FUNCTION_BLOCK FB_Tracking
VAR_IN_OUT
	stAxis  : ARRAY [GVL.cXP .. GVL.cXM] OF ST_AxisGroup;	
END_VAR
VAR_INPUT
	eCommand 			: E_Commands;
	bMotionDone			: BOOL;
	inReset				: ST_Reset;
	inMoveAxisAbsolute	: ST_MoveAxisAbsolute;
	inMoveAxisRelative	: ST_MoveAxisRelative;
END_VAR
VAR_OUTPUT
	stOutMotionDone : ST_MotionDone;
END_VAR
VAR
	//used in tracking Action
	stTrack			: ARRAY [0 .. 4] OF ST_TRACK;
	stTrackTemp		: ST_TRACK;  // Used for the sorting of stTrack.
	keepSorting		: BOOL;      // Used for the sorting.
	bGoNextSeq		: BOOL;
	nAxisID			: INT;
	nMask			: ULINT := 16#FFFF_FFFF_0000_0000;
	
	//used in determining target duration
	fSpeed			: LREAL;
	tTargetDur		: LTIME;
	fDistance		: LREAL;
	
	fbMoving_Rtrig : ARRAY[0 .. 1] OF R_TRIG;
	fbRtrig		: ARRAY[GVL.cHallLower..GVL.cHallUpper] OF R_Trig;
	bInMotion	: BOOL;
	stMotionDone : ARRAY [0..1] OF ST_MotionDone;	
	nSequence	: DINT;
	nLastMoved	: INT;
	
	//counter
	i, j, k, m		: INT := 0;
	nTPC	: INT; //Trip Per Cycle

	// Save task-start and MIO SysTime values in a ring buffer x of depth N. The newest
	// entry is x[i], the oldest is x[(i + 1) mod N], assuming that the buffer is full.
	iTimeBuffer: INT := GVL.cTimeBufferDepth - 1;
	taskStartExtTime: T_TaskStartTimes;
	mioSysTime: T_MioSysTimes;

END_VAR

//////////////////////////////////////////////////////////////
// Call this function block once per cycle to process any updated information about blade set motion and send updates to CCS if required.
//////////////////////////////////////////////////////////////

// Update some times for the previous and current cycles.
iTimeBuffer := (iTimeBuffer + 1) MOD GVL.cTimeBufferDepth;
taskStartExtTime[iTimeBuffer] := F_GetCurExtTime64(GVL.DcToExtTimeOffset, GVL.DcToTcTimeOffset);
mioSysTime[iTimeBuffer] := GVL.mioSysTime;

stAxis[GVL.cXP].bTrackedFlag:=FALSE;
stAxis[GVL.cXM].bTrackedFlag:=FALSE;
nTPC:=0;

// Detect start of motion for the +X blade set, rising edge of its Moving flag from the motor controller.
// Reset motion profile parameters in a local motion-done message not monitored by CCS.
fbMoving_Rtrig[GVL.cXP](CLK:=stAxis[GVL.cXP].axisRef.Status.Moving);
IF fbMoving_Rtrig[GVL.cXP].Q THEN
	// Prepare to record motion profile information.
	bInMotion:=TRUE;  // We're moving!
	stMotionDone[GVL.cXP].axisNum := GVL.cXP; // Axis is +X.
	stMotionDone[GVL.cXP].nsamples := 0;      // No encoder samples yet.
	stMotionDone[GVL.cXP].ntrans := 0;        // No Hall transitions yet.
	stMotionDone[gvl.cXP].startPos := stAxis[GVL.cXP].axisRef.NcToPlc.ActPos;   // Where are we now?
	stMotionDone[GVL.cXP].startTime := taskStartExtTime[iTimeBuffer];
	stMotionDone[GVL.cXP].targetDur := LTIME#0D0H0M0S0MS0US0NS;  // Don't know yet how long this motion will take.
END_IF

// The same, but for the -X blade set.
fbMoving_Rtrig[GVL.cXM](CLK:=stAxis[GVL.cXM].axisRef.Status.Moving);
IF fbMoving_Rtrig[GVL.cXM].Q THEN
	// Prepare to record motion profile information.
	bInMotion:=TRUE;
	stMotionDone[gvl.cXM].axisNum := GVL.cXM;
	stMotionDone[gvl.cXM].nsamples := 0;
	stMotionDone[gvl.cXM].ntrans := 0;
	stMotionDone[gvl.cXM].startPos := stAxis[GVL.cXM].axisRef.NcToPlc.ActPos;
	stMotionDone[gvl.cXM].startTime := taskStartExtTime[iTimeBuffer];
	stMotionDone[gvl.cXM].targetDur := LTIME#0D0H0M0S0MS0US0NS;
END_IF

// Assuming that a motion command was issued by CCS, calculate how long the motion is supposed to last.
// Output is tTargetDur.
IF eCommand = E_Commands.takeExposure THEN
	fSpeed	:= inReset.speed;   // Speed from reset command (actually now set elsewhere in this PLC code).
	IF (fSpeed>0) THEN
		IF (fSpeed>1668.355556) THEN
			fSpeed:=1668.355556;
		END_IF
		tTargetDur 	:= LREAL_TO_LTIME((2*GVL.cPosEnd)/(fSpeed)*EXPT(10,9));
	END_IF
ELSIF eCommand = E_Commands.moveAxisAbsolute THEN
	// MoveAxisAbsolute message contains target position and speed of motion.
	fDistance := ABS(stAxis[inMoveAxisAbsolute.axisIndex].axisRef.NcToPlc.ActPos - inMoveAxisAbsolute.position);
	fSpeed	:= inMoveAxisAbsolute.speed;
	IF (fSpeed>0) THEN
		IF (fSpeed>1668.355556) THEN
			fSpeed:=1668.355556;
		END_IF
		tTargetDur 	:= LREAL_TO_LTIME(((2*fDistance)/(fSpeed))*EXPT(10,9));
	END_IF
ELSIF eCommand = E_Commands.moveAxisRelative THEN
	// MoveAxisRelative message contains position change and how long to take to do it.
	tTargetDur	:= TIME_TO_LTIME(inMoveAxisRelative.moveTime);
END_IF

//Checks to see which blade set last started moving.
IF (stAxis[GVL.cXM].axisRef.Status.Moving AND stAxis[GVL.cXP].axisRef.Status.InTargetPosition) THEN
	nLastMoved:=GVL.cXM;
ELSIF (stAxis[GVL.cXP].axisRef.Status.Moving AND stAxis[GVL.cXM].axisRef.Status.InTargetPosition) THEN
	nLastMoved:=GVL.cXP;
END_IF

////////// Handle the completion of a blade set motion. //////////
IF bMotionDone THEN
	//use for determining which blade set has finished during a travelling slit motion
	IF (stAxis[GVL.cXM].axisRef.Status.Moving AND stAxis[GVL.cXP].axisRef.Status.InTargetPosition) THEN
		nAxisID:=GVL.cXP;
	ELSIF (stAxis[GVL.cXP].axisRef.Status.Moving AND stAxis[GVL.cXM].axisRef.Status.InTargetPosition) THEN
		nAxisID:=GVL.cXM;
	ELSE 
		nAxisID:=nLastMoved;
	END_IF
	//bInMotion flag remains true if either of the blade sets is still in motion
	IF ((NOT stAxis[GVL.cXP].axisRef.Status.Moving) AND (NOT stAxis[GVL.cXM].axisRef.Status.Moving)) THEN
		bInMotion := FALSE;
	END_IF
	// Complete our local motion-done message.
	nSequence := nSequence+1;
	// The motor controller doesn't report exactly when motion was completed, so we assume that it was when the process data
	// from the controller reached us, i.e., at the start of the current cycle.
	stMotionDone[nAxisID].actualDur := ULINT_TO_LTIME(taskStartExtTime[iTimeBuffer] - stMotionDone[nAxisID].startTime);
	stMotionDone[nAxisID].targetDur := tTargetDur;
	stMotionDone[nAxisID].targetPos := stAxis[nAxisID].axisRef.NcToPlc.TargetPos;
	stMotionDone[nAxisID].endPos := stAxis[nAxisID].axisRef.NcToPlc.ActPos;
	stMotionDone[nAxisId].ptpState := MAIN.ptpDiagInfo.PTPState;
	stMotionDone[nAxisId].leapSeconds := MAIN.ptpDiagInfo.CurrentUtcOffset;
	stMotionDone[nAxisId].leapIsValid := TO_BOOL(MAIN.ptpDiagInfo.CurrentUtcOffsetIsValid);
	// Copy our local motion-done message to the location that's monitored by CCS.
	stOutMotionDone:=stMotionDone[nAxisID];
	stOutMotionDone.sequence:=nSequence;  // Ensure message gets sent to CCS by making sure that at least one field has a changed value.
END_IF


////////// Collect information on any Hall switch transitions from the MIOs. //////////
// nNumOfINputs[i] is linked to the event count for the MIO channel assigned to Hall sensor i.
// bInputEventState[i] is linked to the current MIO channel state for Hall sensor i.
// nInputEventTime[i] is linked to the first transition timestamp for Hall sensor i. We assume there is at most one per cycle per channel, though
// more than one channel may have a timestamp available in the same cycle.
// New timestamps are added to the end of the stTrack array.

FOR i:=GVL.cHallLower TO GVL.cHallUpper BY 1 DO
	fbRtrig[i](CLK:=GVL.nNumOfInputs[i].0);  // Look for a rising edge in channel status, which means we have a transition timestamp.
	IF fbRtrig[i].Q THEN
		stTrack[nTPC].nSeqToCompare := INT_TO_WORD((i*10)+5);
		stTrack[nTPC].bEdgeToCompare := GVL.bInputEventState[i];
		stTrack[nTPC].nHallID := i;
		stTrack[nTPC].tScanTime := 
			F_MioExtTime(i, GVL.nInputEventTime[i], iTimeBuffer, taskStartExtTime, mioSysTime);  // ADC timestamp -> ext time.
 		// Count the number of entries stored in stTrack.
		nTPC:=nTPC+1;
	END_IF
END_FOR
	
// Calibration stores events in time order, and later code that assigns locations to Hall events requires
// exactly the same ordering for a given blade set and direction of motion. If during this cycle we picked up
// events from more than one channel we'll have to sort them by time. At most a handful of events
// may occur in a cycle so an exchange sort will do.
IF nTPC > 1 THEN
	keepSorting := TRUE;  // Do we need to keep sorting?
	WHILE keepSorting DO
		keepSorting := FALSE;
		FOR j:= nTPC - 1 TO 1 BY -1 DO
			IF (stTrack[j].tScanTime < stTrack[j-1].tScanTime) THEN  // Use <, not <=, to make it a stable sort.
				stTrackTemp := stTrack[j];
				stTrack[j] := stTrack[j-1];
				stTrack[j-1] := stTrackTemp;
				keepSorting := TRUE;  // Need to keep sorting if an exchange was made.
			END_IF
		END_FOR
	END_WHILE
END_IF


// If we picked up some Hall transitions this cycle, then we need to take position samples (encoder readout).
// We want to check if the position of a blade set at the time of a Hall transition agrees with the
// Hall switch position taken from the last calibration.
IF nTPC>0 THEN
	FOR k:=0 TO nTPC-1 BY 1 DO
		IF (stAxis[GVL.cXP].axisRef.Status.Moving AND stAxis[GVL.cXM].axisRef.Status.Moving) AND
			(stAxis[GVL.cXP].axisRef.Status.PositiveDirection AND stAxis[GVL.cXM].axisRef.Status.PositiveDirection) THEN
			ACT_TrackingDoublePositive();
		ELSIF (stAxis[GVL.cXP].axisRef.Status.Moving AND stAxis[GVL.cXM].axisRef.Status.Moving) AND
			(stAxis[GVL.cXP].axisRef.Status.NegativeDirection AND stAxis[GVL.cXM].axisRef.Status.NegativeDirection) THEN
			ACT_TrackingDoubleNegative();
		ELSE
			ACT_TrackingSingle();
		END_IF
		bGoNextSeq:=FALSE;
	END_FOR
END_IF

ACTION ACT_TrackingDoubleNegative:
// Take encoder samples and compare against Hall transitions when both blade sets are moving toward decreasing camera X coordinate.
// Remember, this code is being called from inside a loop over the contents of stTrack[] with k being the loop variable.
// We have to first assign a Hall event to a blade set before we can find out the motion start times and
// calculate elapsed times from that. 

// +X blade set
IF stAxis[GVL.cXP].axisRef.Status.Moving THEN
	//Compare current sequence with recorded sequence. Update position if match. Negative direction.
	IF stAxis[GVL.cXP].axisRef.status.NegativeDirection AND stAxis[GVL.cXP].stHall[GVL.cDirNeg, stAxis[GVL.cXP].nTripCount].nSeq = stTrack[k].nSeqToCompare AND
			stAxis[GVL.cXP].stHall[GVL.cDirNeg, stAxis[GVL.cXP].nTripCount].bEdge = stTrack[k].bEdgeToCompare AND (NOT bGoNextSeq) THEN
		stAxis[GVL.cXP].fHallPosAct := stAxis[GVL.cXP].fHallPosCal[GVL.cDirNeg, stAxis[GVL.cXP].nTripCount];
		stAxis[GVL.cXP].nTripCount := stAxis[GVL.cXP].nTripCount - 1;		
		//track difference between hall sensor and encoder data at trip point
		stAxis[GVL.cXP].fPosDiffAtTrip := stAxis[GVL.cXP].axisRef.NcToPlc.ActPos - stAxis[GVL.cXP].fHallPosAct;
		stAxis[GVL.cXP].bTrackedFlag:=TRUE;
		bGoNextSeq:=TRUE;
		
		IF bInMotion AND MAIN.outShutterStatus.smState<>E_StatesMaint.Calibrating THEN
			nAxisID := GVL.cXP;
			// The Hall event belongs to the +X blade set.
			stMotionDone[GVL.cXP].trans[stMotionDone[GVL.cXP].ntrans].extTime := stTrack[k].tScanTime;
			stMotionDone[GVL.cXP].trans[stMotionDone[GVL.cXP].ntrans].id := stTrack[k].nHallID;
			stMotionDone[GVL.cXP].trans[stMotionDone[GVL.cXP].ntrans].on := stTrack[k].bEdgeToCompare;
			stMotionDone[GVL.cXP].trans[stMotionDone[GVL.cXP].ntrans].pos := stAxis[GVL.cXP].fHallPosAct;
			stMotionDone[GVL.cXP].ntrans := stMotionDone[GVL.cXP].ntrans +1;
			// We're taking the encoder value from process data for this cycle, so the closest
			// approximation we have to the actual sample time is the time at the start of the cycle.
			stMotionDone[GVL.cXP].samples[stMotionDone[GVL.cXP].nsamples].extTime := taskStartExtTime[iTimeBuffer];
			stMotionDone[GVL.cXP].samples[stMotionDone[GVL.cXP].nsamples].pos := stAxis[GVL.cXP].axisRef.NcToPlc.ActPos;
			stMotionDone[GVL.cXP].nsamples := stMotionDone[GVL.cXP].nsamples + 1;
		END_IF
		
	END_IF
END_IF

// -X blade set
IF stAxis[GVL.cXM].axisRef.Status.Moving THEN
	//Compare current sequence with recorded sequence. Update position if match. Negative direction.
	IF stAxis[GVL.cXM].axisRef.status.NegativeDirection AND stAxis[GVL.cXM].stHall[GVL.cDirNeg, stAxis[GVL.cXM].nTripCount].nSeq = stTrack[k].nSeqToCompare AND
			stAxis[GVL.cXM].stHall[GVL.cDirNeg, stAxis[GVL.cXM].nTripCount].bEdge = stTrack[k].bEdgeToCompare AND (NOT bGoNextSeq) THEN
		stAxis[GVL.cXM].fHallPosAct := stAxis[GVL.cXM].fHallPosCal[GVL.cDirNeg, stAxis[GVL.cXM].nTripCount];
		stAxis[GVL.cXM].nTripCount := stAxis[GVL.cXM].nTripCount + 1;	
		//track difference between hall sensor and encoder data at trip point
		stAxis[GVL.cXM].fPosDiffAtTrip := stAxis[GVL.cXM].axisRef.NcToPlc.ActPos - stAxis[GVL.cXM].fHallPosAct;
		stAxis[GVL.cXM].bTrackedFlag:=TRUE;
		bGoNextSeq:=TRUE;
		
		IF bInMotion AND MAIN.outShutterStatus.smState<>E_StatesMaint.Calibrating THEN
			nAxisID:= GVL.cXM;
			// The Hall event belongs to the -X blade set.
			stMotionDone[GVL.cXM].trans[stMotionDone[GVL.cXM].ntrans].extTime := stTrack[k].tScanTime;
			stMotionDone[GVL.cXM].trans[stMotionDone[GVL.cXM].ntrans].id := stTrack[k].nHallID;
			stMotionDone[GVL.cXM].trans[stMotionDone[GVL.cXM].ntrans].on := stTrack[k].bEdgeToCompare;
			stMotionDone[GVL.cXM].trans[stMotionDone[GVL.cXM].ntrans].pos := stAxis[GVL.cXM].fHallPosAct;
			stMotionDone[GVL.cXM].ntrans := stMotionDone[GVL.cXM].ntrans +1;

			stMotionDone[GVL.cXM].samples[stMotionDone[GVL.cXM].nsamples].extTime := taskStartExtTime[iTimeBuffer];
			stMotionDone[GVL.cXM].samples[stMotionDone[GVL.cXM].nsamples].pos := stAxis[GVL.cXM].axisRef.NcToPlc.ActPos;
			stMotionDone[GVL.cXM].nsamples := stMotionDone[GVL.cXM].nsamples + 1;
		END_IF
		
	END_IF
END_IF
END_ACTION

ACTION ACT_TrackingDoublePositive:
// Take encoder samples and compare against Hall transitions when both blade sets are moving toward increasing camera X coordinate.

// -X blade set
IF stAxis[GVL.cXM].axisRef.Status.Moving THEN
	//Compare current sequence with recorded sequence. Update position if match. Positive direction.
	IF stAxis[GVL.cXM].axisRef.status.PositiveDirection AND stAxis[GVL.cXM].stHall[GVL.cDirPos, stAxis[GVL.cXM].nTripCount].nSeq = stTrack[k].nSeqToCompare AND
			stAxis[GVL.cXM].stHall[GVL.cDirPos, stAxis[GVL.cXM].nTripCount].bEdge = stTrack[k].bEdgeToCompare AND (NOT bGoNextSeq) THEN
		stAxis[GVL.cXM].fHallPosAct := stAxis[GVL.cXM].fHallPosCal[GVL.cDirPos, stAxis[GVL.cXM].nTripCount];
		stAxis[GVL.cXM].nTripCount := stAxis[GVL.cXM].nTripCount - 1;	
		//track difference between hall sensor and encoder data at trip point
		stAxis[GVL.cXM].fPosDiffAtTrip := stAxis[GVL.cXM].axisRef.NcToPlc.ActPos - stAxis[GVL.cXM].fHallPosAct;
		stAxis[GVL.cXM].bTrackedFlag:=TRUE;
		bGoNextSeq:=TRUE;
		
		IF bInMotion AND MAIN.outShutterStatus.smState<>E_StatesMaint.Calibrating THEN
			nAxisID:= GVL.cXM;
			// The Hall event belongs to the -X blade set.
			stMotionDone[GVL.cXM].trans[stMotionDone[GVL.cXM].ntrans].extTime := stTrack[k].tScanTime;
			stMotionDone[GVL.cXM].trans[stMotionDone[GVL.cXM].ntrans].id := stTrack[k].nHallID;
			stMotionDone[GVL.cXM].trans[stMotionDone[GVL.cXM].ntrans].on := stTrack[k].bEdgeToCompare;
			stMotionDone[GVL.cXM].trans[stMotionDone[GVL.cXM].ntrans].pos := stAxis[GVL.cXM].fHallPosAct;
			stMotionDone[GVL.cXM].ntrans := stMotionDone[GVL.cXM].ntrans +1;
			
			stMotionDone[GVL.cXM].samples[stMotionDone[GVL.cXM].nsamples].extTime := taskStartExtTime[iTimeBuffer];
			stMotionDone[GVL.cXM].samples[stMotionDone[GVL.cXM].nsamples].pos := stAxis[GVL.cXM].axisRef.NcToPlc.ActPos;
			stMotionDone[GVL.cXM].nsamples := stMotionDone[GVL.cXM].nsamples + 1;
		END_IF
		
	END_IF
END_IF

// +X blade set
IF stAxis[GVL.cXP].axisRef.Status.Moving THEN
	//Compare current sequence with recorded sequence. Update position if match. Positive direction.
	IF stAxis[GVL.cXP].axisRef.status.PositiveDirection AND stAxis[GVL.cXP].stHall[GVL.cDirPos, stAxis[GVL.cXP].nTripCount].nSeq = stTrack[k].nSeqToCompare AND 
			stAxis[GVL.cXP].stHall[GVL.cDirPos, stAxis[GVL.cXP].nTripCount].bEdge = stTrack[k].bEdgeToCompare AND (NOT bGoNextSeq) THEN
		stAxis[GVL.cXP].fHallPosAct := stAxis[GVL.cXP].fHallPosCal[GVL.cDirPos, stAxis[GVL.cXP].nTripCount];
		stAxis[GVL.cXP].nTripCount := stAxis[GVL.cXP].nTripCount + 1;
		//track difference between hall sensor and encoder data at trip point
		stAxis[GVL.cXP].fPosDiffAtTrip := stAxis[GVL.cXP].axisRef.NcToPlc.ActPos - stAxis[GVL.cXP].fHallPosAct;
		stAxis[GVL.cXP].bTrackedFlag:=TRUE;
		bGoNextSeq:=TRUE;
		
		IF bInMotion AND MAIN.outShutterStatus.smState<>E_StatesMaint.Calibrating THEN
			nAxisID:= GVL.cXP;
			// The Hall event belongs to the +X blade set.
			stMotionDone[GVL.cXP].trans[stMotionDone[GVL.cXP].ntrans].extTime := stTrack[k].tScanTime;
			stMotionDone[GVL.cXP].trans[stMotionDone[GVL.cXP].ntrans].id := stTrack[k].nHallID;
			stMotionDone[GVL.cXP].trans[stMotionDone[GVL.cXP].ntrans].on := stTrack[k].bEdgeToCompare;
			stMotionDone[GVL.cXP].trans[stMotionDone[GVL.cXP].ntrans].pos := stAxis[GVL.cXP].fHallPosAct;
			stMotionDone[GVL.cXP].ntrans := stMotionDone[GVL.cXP].ntrans +1;
			
			// We're taking the encoder value from process data for this cycle, so the closest
			// approximation we have to the actual sample time is the time at the start of the cycle.
			stMotionDone[GVL.cXP].samples[stMotionDone[GVL.cXP].nsamples].extTime := taskStartExtTime[iTimeBuffer];
			stMotionDone[GVL.cXP].samples[stMotionDone[GVL.cXP].nsamples].pos := stAxis[GVL.cXP].axisRef.NcToPlc.ActPos;
			stMotionDone[GVL.cXP].nsamples := stMotionDone[GVL.cXP].nsamples + 1;
		END_IF
		
	END_IF
END_IF
END_ACTION

ACTION ACT_TrackingSingle:
// Take encoder samples and compare against Hall transitions when only one blade set is moving.

// +X blade set
IF stAxis[GVL.cXP].axisRef.Status.Moving THEN
	//Compare current sequence with recorded sequence. Update position if match. Positive direction.
	IF stAxis[GVL.cXP].axisRef.status.PositiveDirection AND stAxis[GVL.cXP].stHall[GVL.cDirPos, stAxis[GVL.cXP].nTripCount].nSeq = stTrack[k].nSeqToCompare AND 
			stAxis[GVL.cXP].stHall[GVL.cDirPos, stAxis[GVL.cXP].nTripCount].bEdge = stTrack[k].bEdgeToCompare AND (NOT bGoNextSeq) THEN
		stAxis[GVL.cXP].fHallPosAct := stAxis[GVL.cXP].fHallPosCal[GVL.cDirPos, stAxis[GVL.cXP].nTripCount];
		stAxis[GVL.cXP].nTripCount := stAxis[GVL.cXP].nTripCount + 1;
		//track difference between hall sensor and encoder data at trip point
		stAxis[GVL.cXP].fPosDiffAtTrip := stAxis[GVL.cXP].axisRef.NcToPlc.ActPos - stAxis[GVL.cXP].fHallPosAct;
		stAxis[GVL.cXP].bTrackedFlag:=TRUE;
		bGoNextSeq:=TRUE;
		
		IF bInMotion AND MAIN.outShutterStatus.smState<>E_StatesMaint.Calibrating THEN
			nAxisID:= GVL.cXP;
			// The Hall event belongs to the +X blade set.
			stMotionDone[GVL.cXP].trans[stMotionDone[GVL.cXP].ntrans].extTime := stTrack[k].tScanTime;
			stMotionDone[GVL.cXP].trans[stMotionDone[GVL.cXP].ntrans].id := stTrack[k].nHallID;
			stMotionDone[GVL.cXP].trans[stMotionDone[GVL.cXP].ntrans].on := stTrack[k].bEdgeToCompare;
			stMotionDone[GVL.cXP].trans[stMotionDone[GVL.cXP].ntrans].pos := stAxis[GVL.cXP].fHallPosAct;
			stMotionDone[GVL.cXP].ntrans := stMotionDone[GVL.cXP].ntrans +1;			
			// We're taking the encoder value from process data for this cycle, so the closest
			// approximation we have to the actual sample time is the time at the start of the cycle.
			stMotionDone[GVL.cXP].samples[stMotionDone[GVL.cXP].nsamples].extTime := taskStartExtTime[iTimeBuffer];
			stMotionDone[GVL.cXP].samples[stMotionDone[GVL.cXP].nsamples].pos := stAxis[GVL.cXP].axisRef.NcToPlc.ActPos;
			stMotionDone[GVL.cXP].nsamples := stMotionDone[GVL.cXP].nsamples + 1;
		END_IF
		
	END_IF
	//Compare current sequence with recorded sequence. Update position if match. Negative direction.
	IF stAxis[GVL.cXP].axisRef.status.NegativeDirection AND stAxis[GVL.cXP].stHall[GVL.cDirNeg, stAxis[GVL.cXP].nTripCount].nSeq = stTrack[k].nSeqToCompare AND
			stAxis[GVL.cXP].stHall[GVL.cDirNeg, stAxis[GVL.cXP].nTripCount].bEdge = stTrack[k].bEdgeToCompare AND (NOT bGoNextSeq) THEN
		stAxis[GVL.cXP].fHallPosAct := stAxis[GVL.cXP].fHallPosCal[GVL.cDirNeg, stAxis[GVL.cXP].nTripCount];
		stAxis[GVL.cXP].nTripCount := stAxis[GVL.cXP].nTripCount - 1;		
		//track difference between hall sensor and encoder data at trip point
		stAxis[GVL.cXP].fPosDiffAtTrip := stAxis[GVL.cXP].axisRef.NcToPlc.ActPos - stAxis[GVL.cXP].fHallPosAct;
		stAxis[GVL.cXP].bTrackedFlag:=TRUE;
		bGoNextSeq:=TRUE;
		
		IF bInMotion AND MAIN.outShutterStatus.smState<>E_StatesMaint.Calibrating THEN
			nAxisID:= GVL.cXP;
			// The Hall event belongs to the +X blade set.
			stMotionDone[GVL.cXP].trans[stMotionDone[GVL.cXP].ntrans].extTime := stTrack[k].tScanTime;
			stMotionDone[GVL.cXP].trans[stMotionDone[GVL.cXP].ntrans].id := stTrack[k].nHallID;
			stMotionDone[GVL.cXP].trans[stMotionDone[GVL.cXP].ntrans].on := stTrack[k].bEdgeToCompare;
			stMotionDone[GVL.cXP].trans[stMotionDone[GVL.cXP].ntrans].pos := stAxis[GVL.cXP].fHallPosAct;
			stMotionDone[GVL.cXP].ntrans := stMotionDone[GVL.cXP].ntrans +1;
			
			stMotionDone[GVL.cXP].samples[stMotionDone[GVL.cXP].nsamples].extTime := taskStartExtTime[iTimeBuffer];
			stMotionDone[GVL.cXP].samples[stMotionDone[GVL.cXP].nsamples].pos := stAxis[GVL.cXP].axisRef.NcToPlc.ActPos;
			stMotionDone[GVL.cXP].nsamples := stMotionDone[GVL.cXP].nsamples + 1;
		END_IF
		
	END_IF
END_IF

// -X blade set
IF stAxis[GVL.cXM].axisRef.Status.Moving THEN
	//Compare current sequence with recorded sequence. Update position if match. Positive direction.
	IF stAxis[GVL.cXM].axisRef.status.PositiveDirection AND stAxis[GVL.cXM].stHall[GVL.cDirPos, stAxis[GVL.cXM].nTripCount].nSeq = stTrack[k].nSeqToCompare AND
			stAxis[GVL.cXM].stHall[GVL.cDirPos, stAxis[GVL.cXM].nTripCount].bEdge = stTrack[k].bEdgeToCompare AND (NOT bGoNextSeq) THEN
		stAxis[GVL.cXM].fHallPosAct := stAxis[GVL.cXM].fHallPosCal[GVL.cDirPos, stAxis[GVL.cXM].nTripCount];
		stAxis[GVL.cXM].nTripCount := stAxis[GVL.cXM].nTripCount - 1;	
		//track difference between hall sensor and encoder data at trip point
		stAxis[GVL.cXM].fPosDiffAtTrip := stAxis[GVL.cXM].axisRef.NcToPlc.ActPos - stAxis[GVL.cXM].fHallPosAct;
		stAxis[GVL.cXM].bTrackedFlag:=TRUE;
		bGoNextSeq:=TRUE;
		
		IF bInMotion AND MAIN.outShutterStatus.smState<>E_StatesMaint.Calibrating THEN
			nAxisID:= GVL.cXM;
			// The Hall event belongs to the -X blade set.
			stMotionDone[GVL.cXM].trans[stMotionDone[GVL.cXM].ntrans].extTime := stTrack[k].tScanTime;
			stMotionDone[GVL.cXM].trans[stMotionDone[GVL.cXM].ntrans].id := stTrack[k].nHallID;
			stMotionDone[GVL.cXM].trans[stMotionDone[GVL.cXM].ntrans].on := stTrack[k].bEdgeToCompare;
			stMotionDone[GVL.cXM].trans[stMotionDone[GVL.cXM].ntrans].pos := stAxis[GVL.cXM].fHallPosAct;
			stMotionDone[GVL.cXM].ntrans := stMotionDone[GVL.cXM].ntrans +1;
			
			stMotionDone[GVL.cXM].samples[stMotionDone[GVL.cXM].nsamples].extTime := taskStartExtTime[iTimeBuffer];
			stMotionDone[GVL.cXM].samples[stMotionDone[GVL.cXM].nsamples].pos := stAxis[GVL.cXM].axisRef.NcToPlc.ActPos;
			stMotionDone[GVL.cXM].nsamples := stMotionDone[GVL.cXM].nsamples + 1;
		END_IF
		
	END_IF
	//Compare current sequence with recorded sequence. Update position if match. Negative direction.
	IF stAxis[GVL.cXM].axisRef.status.NegativeDirection AND stAxis[GVL.cXM].stHall[GVL.cDirNeg, stAxis[GVL.cXM].nTripCount].nSeq = stTrack[k].nSeqToCompare AND
			stAxis[GVL.cXM].stHall[GVL.cDirNeg, stAxis[GVL.cXM].nTripCount].bEdge = stTrack[k].bEdgeToCompare AND (NOT bGoNextSeq) THEN
		stAxis[GVL.cXM].fHallPosAct := stAxis[GVL.cXM].fHallPosCal[GVL.cDirNeg, stAxis[GVL.cXM].nTripCount];
		stAxis[GVL.cXM].nTripCount := stAxis[GVL.cXM].nTripCount + 1;	
		//track difference between hall sensor and encoder data at trip point
		stAxis[GVL.cXM].fPosDiffAtTrip := stAxis[GVL.cXM].axisRef.NcToPlc.ActPos - stAxis[GVL.cXM].fHallPosAct;
		stAxis[GVL.cXM].bTrackedFlag:=TRUE;
		bGoNextSeq:=TRUE;
		
		IF bInMotion AND MAIN.outShutterStatus.smState<>E_StatesMaint.Calibrating THEN
			nAxisID:= GVL.cXM;
			// The Hall event belongs to the -X blade set.
			stMotionDone[GVL.cXM].trans[stMotionDone[GVL.cXM].ntrans].extTime := stTrack[k].tScanTime;
			stMotionDone[GVL.cXM].trans[stMotionDone[GVL.cXM].ntrans].id := stTrack[k].nHallID;
			stMotionDone[GVL.cXM].trans[stMotionDone[GVL.cXM].ntrans].on := stTrack[k].bEdgeToCompare;
			stMotionDone[GVL.cXM].trans[stMotionDone[GVL.cXM].ntrans].pos := stAxis[GVL.cXM].fHallPosAct;
			stMotionDone[GVL.cXM].ntrans := stMotionDone[GVL.cXM].ntrans +1;
			
			stMotionDone[GVL.cXM].samples[stMotionDone[GVL.cXM].nsamples].extTime := taskStartExtTime[iTimeBuffer];
			stMotionDone[GVL.cXM].samples[stMotionDone[GVL.cXM].nsamples].pos := stAxis[GVL.cXM].axisRef.NcToPlc.ActPos;
			stMotionDone[GVL.cXM].nsamples := stMotionDone[GVL.cXM].nsamples + 1;
		END_IF
		
	END_IF
END_IF
END_ACTION

END_FUNCTION_BLOCK

(* stored: Version 1.1.0.1, ProductVersion 3.1.4022.18
   POU FB_Tracking: Id {462a5933-fe60-42d4-a574-27170521c4c5}, SpecialFunc None
   Action ACT_TrackingDoubleNegative: Id {0039cb21-b703-43f6-867c-8fbe57c73e86}
   Action ACT_TrackingDoublePositive: Id {015fe346-39d0-42ba-a488-79403589a261}
   Action ACT_TrackingSingle: Id {68bb727f-4301-4350-9f19-54a85b8d6b0c} *)
